// TIA Portal V20 export
// export: Created 2026-07-10T11:12:32.753665Z, ExportSetting WithDefaults, DisplayName Totally Integrated Automation Portal, DisplayVersion V20, DisplayName TIA Portal Openness, DisplayVersion V20, DisplayName TIA Portal Version Control Interface, DisplayVersion V20, DisplayName STEP 7 Professional, DisplayVersion V20, DisplayName STEP 7 Safety, DisplayVersion V20, DisplayName WinCC Basic/Comfort/Advanced, DisplayVersion V20, DisplayName WinCC Unified, DisplayVersion V20
FUNCTION_BLOCK "DamperController"   // FB8, SCL
{ S7_Optimized_Access := 'TRUE' }
VERSION : 0.1
// stored: AutoNumber true, IsIECCheckEnabled false, IsRetainMemResEnabled false, MemoryReserve 100, SetENOAutomatically false, UDAEnableTagReadback false
   VAR_INPUT
      ManualMode : Bool;
      ManaulOpen : Bool;
      ManualClose : Bool;
      TankLevel : Real;
      TankLevelSetpoint : Real;
      TankLevelMin : Real;
      TankLevelMax : Real;
      UsePID : Bool;
      PID_DeadZone : Real;
      PID_KP : Real;
      PID_KI : Real;
      PID_KD : Real;
      PID_TI : Real;
      LimitSwitch0 : Bool;
      LimitSwitch100 : Bool;
      PouseMove : UInt := 10;
      PositionDeadzone : Real := 1.0;
      StartAjustment : Bool;
      CancelAjustment : Bool;
      ResetPosition : Bool;
      SwitchAutoMode : Bool;
   END_VAR
   VAR_OUTPUT
      Open : Bool;
      Close : Bool;
      CurrentPosition : Real;
      PositionError : Bool;
      PositionSetPoint : Real;
      AdjustBusy : Bool;
      AdjustError : Bool;
   END_VAR
   VAR_IN_OUT
      FullMovingTime : Real;
   END_VAR
   VAR
      MoveToLimitSwitch : Bool;
      AdjustmentDone : Word;
      LappedSetpoint : Real;
      isMoving : Bool;
      isAutoMode : Bool;
      isReady : Bool;
      EnablePIDTON { S7_SetPoint := 'True'} : TON_TIME;
      PIDRegulator { S7_SetPoint := 'True'} : "PIDRegulator";
      HystRegulator { S7_SetPoint := 'True'} : "HystRegulator";
      RepositionRTrig { S7_SetPoint := 'True'} : R_TRIG;
      MotorPositionNoFeedback { S7_SetPoint := 'True'} : "MotorPositionNoFeedback";
      MotorController { S7_SetPoint := 'True'} : "MotorControllerSimple";
      RepositionTON { S7_SetPoint := 'True'} : TON_TIME;
      MotorMoverToSwitch { S7_SetPoint := 'True'} : "MotorMoverToSwitch";
      MotorAdjustmentNoFeedback { S7_SetPoint := 'True'} : "MotorAdjustmentNoFeedback";
   END_VAR
   VAR CONSTANT
      LappingZone0 : Real := 1.0;
      LappingZone100 : Real := 2.0;
      EnablePIDTime : Time := T#10s;
   END_VAR
BEGIN
   #isMoving := #Open OR #Close;
   #isAutoMode := NOT #ManualMode;
   #isReady := #isAutoMode;

   #EnablePIDTON(IN:=#UsePID AND #isReady,
                 PT:= #EnablePIDTime);

   #PIDRegulator(Enable:=#EnablePIDTON.Q,
                 Tanklevel:=#TankLevel,
                 TankLevelSetpoint:=#TankLevelSetpoint,
                 KP:=#PID_KP,
                 KI:=#PID_KI,
                 KD:=#PID_KD,
                 TI:=DINT_TO_TIME(REAL_TO_DINT(#PID_TI)*1000),
                 LimitMin:=0,
                 DeadZone := #PID_DeadZone);


   #PositionSetPoint := LIMIT(MN := 0, IN := #PIDRegulator.DamperPosition, MX := 100);

   IF #TankLevel > #TankLevelMax THEN
       #PositionSetPoint := 0;
   END_IF;

   IF #TankLevel < #TankLevelMin THEN
       #PositionSetPoint := 100;
   END_IF;

   #HystRegulator(Enable:=#isAutoMode AND (NOT #UsePID),
                  TankLevel:=#TankLevel,
                  TankLevelMin:=#TankLevelMin,
                  TankLevelMax:=#TankLevelMax);

   #RepositionRTrig(CLK:=#ResetPosition);

   #MotorPositionNoFeedback(Enable:=TRUE,
                            LimitSwitch0:=#LimitSwitch0,
                            LimitSwitch100:=#LimitSwitch100,
                            Invalidate:=#RepositionRTrig.Q,
                            FullMovingTime:=#FullMovingTime,
                            LappingZone:=#PositionDeadzone,
                            Open:=#Open,
                            Close:=#Close,
                            CurrentPosition=>#CurrentPosition,
                            Error=>#PositionError,
                            SwitchAutoMode := #SwitchAutoMode);

   #LappedSetpoint := #PositionSetPoint;
   IF #PositionSetPoint <= #LappingZone0 THEN
       #LappedSetpoint := 0;
   ELSIF #PositionSetPoint >= (100 - #LappingZone100) THEN
       #LappedSetpoint := 100;
   END_IF;

   #MotorController(Enable := #isAutoMode AND #UsePID,
                    CurrentPosition := #CurrentPosition,
                    SetpointPosition := #LappedSetpoint,
                    PositionDeadzone := #PositionDeadzone,
                    MinimalPulse := REAL_TO_DINT(LIMIT(MN := 0.1, IN := #FullMovingTime / 100, MX := 0.5) * 1000),
                    PauseMode := UINT_TO_TIME(IN := #PouseMove) * 1000,
                    isMoving := #isMoving,
                    MoveNow := FALSE,
                    MinReversPause := T#2s,
                    PositionError:=#PositionError);


   #RepositionTON(IN:=TRUE,
                  PT:=T#10s);

   #MotorMoverToSwitch(Enable:=#RepositionTON.Q,
                       Go:= #PositionError,
                       TargetSwitch100:=FALSE,
                       MovePause:=T#5s,
                       isMoving:=#isMoving,
                       LimitSwitch0:=#LimitSwitch0,
                       LimitSwitch100:=#LimitSwitch100);

   #MotorAdjustmentNoFeedback(Enable:=#isAutoMode,
                              Start:=#StartAjustment,
                              Cancel:=#CancelAjustment,
                              AbortTime:=T#120s,
                              MovePause:=T#5s,
                              isMoving:=#isMoving,
                              LimitSwitch0:=#LimitSwitch0,
                              LimitSwitch100:=#LimitSwitch100,
                              Done:=#AdjustmentDone,
                              FullMovingTime:=#FullMovingTime,
                              Busy => #AdjustBusy,
                              Error => #AdjustError);

   IF ("MB".Table.Alarms_NoPowerSupply OR NOT #SwitchAutoMode) THEN
       #Open := FALSE;
       #Close := FALSE;
       RETURN;
   END_IF;

   IF #ManualMode THEN
       #Open := #ManaulOpen;
       #Close := #ManualClose;

   ELSIF #MotorAdjustmentNoFeedback.Busy THEN
       #Open := #MotorAdjustmentNoFeedback.Open;
       #Close := #MotorAdjustmentNoFeedback.Close;

   ELSIF #PositionError THEN
       #Open := #MotorMoverToSwitch.Open;
       #Close := #MotorMoverToSwitch.Close;

   ELSIF #UsePID THEN
       #Open := #MotorController.Open;
       #Close := #MotorController.Close;
   ELSE
       #Open := #HystRegulator.Open;
       #Close := #HystRegulator.Close;
       #PositionSetPoint := #HystRegulator.PositionSetpoint;
   END_IF;
END_FUNCTION_BLOCK
